TYPE ST_RecipeParam :
STRUCT

	(*Paramètres production*)
	lrPositionBasse: LREAL;
	lrVitesse: LREAL;
	
END_STRUCT
END_TYPE

(* stored: Version 1.1.0.1, ProductVersion 3.1.4020.12
   DUT ST_RecipeParam: Id {0f620af8-c30d-4af7-b0a2-88c84a465146} *)
